(* IEC 61131-3 sources: plc_generation_empirical_study/datasets/packages/internal_v0_1/qualification_only/C02_E01_basic_start_stop_latch, 1 file *)

(* ---- reference.st ---- *)
FUNCTION_BLOCK C02_E01_basic_start_stop_latch
VAR_INPUT
    Start : BOOL;
    Stop : BOOL;
END_VAR
VAR_OUTPUT
    Running : BOOL;
END_VAR

IF Stop THEN
    Running := FALSE;
ELSIF Start THEN
    Running := TRUE;
END_IF;

END_FUNCTION_BLOCK
